// TIA Portal V20 export
DATA_BLOCK "DB_OPC_Components"   // DB118
{ S7_Optimized_Access := 'TRUE' }
// stored: MemoryReserve 100
   VAR
      Backwalls : Struct
         LoaderDrilled : Byte;
         LoaderUndrilled : Byte;
         Shuttle2Drilled : Byte;
         Shuttle2Undrilled : Byte;
         ShuttleDrilled : Byte;
         ShuttleUndrilled : Byte;
         WorkClamp : Byte;
      END_STRUCT;
      Parts : Struct
         LoaderDrilled : Byte;
         LoaderUndrilled : Byte;
         Shuttle2Drilled : Byte;
         Shuttle2Undrilled : Byte;
         ShuttleDrilled : Byte;
         ShuttleUndrilled : Byte;
         WorkClamp : Byte;
      END_STRUCT;
      Update : Byte;
   END_VAR
BEGIN
END_DATA_BLOCK
